FUNCTION_BLOCK FB_Event IMPLEMENTS I_Event
VAR_INPUT
END_VAR
VAR_OUTPUT
END_VAR
VAR
	fbList:				FB_ListString;
	iParent:			I_Component;
	iLogger:			I_Logger;
	stAbort:			ST_Event;
	stStop:				ST_Event;	
	stStopCycle:		ST_Event;
	stWarning:			ST_Event;
	stInformation:		ST_Event;
	stDebug:			ST_Event;
END_VAR

METHOD FB_init : BOOL
VAR_INPUT
	bInitRetains : BOOL; // if TRUE, the retain variables are initialized (warm start / cold start)
	bInCopyCode : BOOL;  // if TRUE, the instance afterwards gets moved into the copy code (online change)
	iParent:			I_Component;
END_VAR
THIS^.iParent:= iParent;
END_METHOD

METHOD PUBLIC M_Abort : BOOL
VAR_INPUT
	Message:				STRING(255);
	ID:						ID;
END_VAR
stAbort.Source:= iParent;
stAbort.Instance:= iParent.P_Info.P_Instance;
stAbort.Class:= iParent.P_Info.P_Class;
stAbort.EventType:= E_Event.Error;
stAbort.Timestamp:= F_GetSystemTime();
stAbort.ID:= ID;
stAbort.Message:= Message;
stAbort.Arguments:= M_Arguments();
stAbort.Command:= 'Abort';
stAbort.Active:= TRUE;

iParent.M_Request(E_Request.Abort);
IF iLogger <> 0 THEN
	iLogger.M_Log(stAbort);
ELSE
	fbLogger.M_Log(stAbort);
END_IF
END_METHOD

METHOD PUBLIC M_AddBOOL
VAR_INPUT
	Value: 	bool;
END_VAR
fbList.M_Add(BOOL_TO_STRING(Value));
END_METHOD

METHOD PUBLIC M_AddINT
VAR_INPUT
	Value: 	LINT;
END_VAR
fbList.M_Add(LINT_TO_STRING(Value));
END_METHOD

METHOD PUBLIC M_AddREAL
VAR_INPUT
	Value: 	Lreal;
	Decimals: INT;
END_VAR
fbList.M_Add(LREAL_TO_FMTSTR(Value, Decimals, TRUE));
END_METHOD

METHOD PUBLIC M_AddSTRING
VAR_INPUT
	Value: STRING(255);
END_VAR
fbList.M_Add(Value);
END_METHOD

METHOD PUBLIC M_AddTIME
VAR_INPUT
	Value: 	TIME;
END_VAR
fbList.M_Add(TIME_TO_STRING(Value));
END_METHOD

METHOD INTERNAL M_Arguments : STRING(255)
VAR_INPUT
END_VAR
VAR
	nIndex:			INT;
END_VAR
WHILE nIndex < fbList. P_Length DO
	M_Arguments:= Concat(Concat(M_Arguments, fbList.M_Index(nIndex)), '$N');
	nIndex:= nIndex + 1;
END_WHILE

fbList.M_Clear();
END_METHOD

METHOD PUBLIC M_Debug : BOOL
VAR_INPUT
	Message:				STRING(255);
END_VAR
stDebug.Source:= iParent;
stDebug.Instance:= iParent.P_Info.P_Instance;
stDebug.Class:= iParent.P_Info.P_Class;
stDebug.EventType:= E_Event.Debug;
stDebug.Timestamp:= F_GetSystemTime();
stDebug.ID:= '';
stDebug.Message:= Message;
stDebug.Arguments:= M_Arguments();
stDebug.Command:= '';
stDebug.Active:= TRUE;

IF iLogger <> 0 THEN
	iLogger.M_Log(stDebug);
ELSE
	fbLogger.M_Log(stDebug);
END_IF
END_METHOD

METHOD PUBLIC M_Information : BOOL
VAR_INPUT
	Message:				STRING(255);
	ID:						ID;
END_VAR
stInformation.Source:= iParent;
stInformation.Instance:= iParent.P_Info.P_Instance;
stInformation.Class:= iParent.P_Info.P_Class;
stInformation.EventType:= E_Event.Information;
stInformation.Timestamp:= F_GetSystemTime();
stInformation.ID:= ID;
stInformation.Message:= Message;
stInformation.Arguments:= M_Arguments();
stInformation.Command:= 'Information';
stInformation.Active:= TRUE;

IF iLogger <> 0 THEN
	iLogger.M_Log(stInformation);
ELSE
	fbLogger.M_Log(stInformation);
END_IF
END_METHOD

METHOD PUBLIC M_Reset
VAR_INPUT
END_VAR
Memset(ADR(stAbort), 0, SIZEOF(stAbort));
Memset(ADR(stStop), 0, SIZEOF(stStop));
Memset(ADR(stStopCycle), 0, SIZEOF(stStopCycle));
Memset(ADR(stWarning), 0, SIZEOF(stWarning));
Memset(ADR(stInformation), 0, SIZEOF(stInformation));
Memset(ADR(stDebug), 0, SIZEOF(stDebug));
END_METHOD

METHOD PUBLIC M_Stop : BOOL
VAR_INPUT
	Message:				STRING(255);
	ID:						ID;
END_VAR
stStop.Source:= iParent;
stStop.Instance:= iParent.P_Info.P_Instance;
stStop.Class:= iParent.P_Info.P_Class;
stStop.EventType:= E_Event.Error;
stStop.Timestamp:= F_GetSystemTime();
stStop.ID:= ID;
stStop.Message:= Message;
stStop.Arguments:= M_Arguments();
stStop.Command:= 'Stop';
stStop.Active:= TRUE;

iParent.M_Request(E_Request.Stop);
IF iLogger <> 0 THEN
	iLogger.M_Log(stStop);
ELSE
	fbLogger.M_Log(stStop);
END_IF
END_METHOD

METHOD PUBLIC M_StopCycle : BOOL
VAR_INPUT
	Message:				STRING(255);
	ID:						ID;
END_VAR
stStopCycle.Source:= iParent;
stStopCycle.Instance:= iParent.P_Info.P_Instance;
stStopCycle.Class:= iParent.P_Info.P_Class;
stStopCycle.EventType:= E_Event.Error;
stStopCycle.Timestamp:= F_GetSystemTime();
stStopCycle.ID:= ID;
stStopCycle.Message:= Message;
stStopCycle.Arguments:= M_Arguments();
stStopCycle.Command:= 'StopCycle';
stStopCycle.Active:= TRUE;

iParent.M_Request(E_Request.StopCycle);
IF iLogger <> 0 THEN
	iLogger.M_Log(stStopCycle);
ELSE
	fbLogger.M_Log(stStopCycle);
END_IF
END_METHOD

METHOD PUBLIC M_Warning : BOOL
VAR_INPUT
	Message:				STRING(255);
	ID:						ID;
END_VAR
stWarning.Source:= iParent;
stWarning.Instance:= iParent.P_Info.P_Instance;
stWarning.Class:= iParent.P_Info.P_Class;
stWarning.EventType:= E_Event.Warning;
stWarning.Timestamp:= F_GetSystemTime();
stWarning.ID:= ID;
stWarning.Message:= Message;
stWarning.Arguments:= M_Arguments();
stWarning.Command:= '';
stWarning.Active:= TRUE;

IF iLogger<> 0 THEN
	iLogger.M_Log(stWarning);
ELSE
	fbLogger.M_Log(stWarning);
END_IF
END_METHOD

PROPERTY PUBLIC P_Logger : I_Logger
GET
P_Logger:= iLogger;
END_GET
SET
iLogger:= P_Logger;
END_SET
END_PROPERTY

END_FUNCTION_BLOCK

(* stored: Version 1.1.0.1
   POU FB_Event: Id {59616103-7f2e-4b6f-81bd-583969a36d28}, SpecialFunc None
   Method FB_init: Id {be23ffcc-529d-4010-ace3-b17baed191a5}
   Method M_Abort: Id {55348828-4763-4c06-9dd1-090fa29a8379}
   Method M_AddBOOL: Id {55367f5b-ac71-0a63-095c-881721842948}
   Method M_AddINT: Id {77c01fd5-65e9-07ed-2cff-a79b9d444c15}
   Method M_AddREAL: Id {b0c25678-4933-0839-34f0-c4eb0def69fb}
   Method M_AddSTRING: Id {8ae81d27-cb47-01bb-2b19-fe8608e777a8}
   Method M_AddTIME: Id {a7c2a656-d860-0eb9-0cff-1e8b5b1d8573}
   Method M_Arguments: Id {70779266-7b36-4bce-9e6f-049e951fd75a}
   Method M_Debug: Id {0a2b992b-2a4a-0251-0210-713b326debf6}
   Method M_Information: Id {d9a244f2-1d6f-434f-aab4-cad6aacbb94f}
   Method M_Reset: Id {31d9e5bb-2957-4381-81b6-d0453bdac8d3}
   Method M_Stop: Id {648ad3fe-ab2e-0b8d-0134-eed394027742}
   Method M_StopCycle: Id {2670afd0-b3e6-08da-2c9f-30a65f88768a}
   Method M_Warning: Id {d443b8bb-774e-487e-80a2-79cf66a0376c}
   Property P_Logger: Id {642d0edf-ded0-4248-be29-8384d3180124}
   Get Get: Id {99e41819-eb78-4b29-b3e9-6728532b14b1}
   Set Set: Id {be31597a-6e88-476b-aec8-980317d6bc1a} *)
